TYPE ST_CycleData :
STRUCT
//-----------------------------------------------------------------------------------GENERAL------------------------------------------------------------------------------------//	

	nNest				: INT;
	bPass				: BOOL;
	bFail				: BOOL;	
	sDate				: STRING;	
	sTime				: STRING;
	
	LeakTest_Pass		: BOOL;
	LeakTest_Fail		: BOOL;
	
	Camera_Pass			: BOOL;
	Camera_Fail			: BOOL;
	
	//Height test
	
	LSS_ScaledHeight			: ARRAY [1..4] OF REAL;
	LSS_anSetPoint				: REAL;
	LSS_CalibrationHeight		: ARRAY [1..4] OF REAL;
	LSS_anRawMeasurement		: ARRAY [1..4] OF REAL;
	LSS_HeightPass				: ARRAY [1..4] OF BOOL;	
	LSS_HeightFail				: ARRAY [1..4] OF BOOL;	

	
	LSS_Pass			: BOOL;
	LSS_Fail			: BOOL;	

	
	//HMI, CSV
	sGeneralResult		: STRING;
	sCameraResult		: STRING;
	sHeightTestResult	: STRING;
	sLeakTesterResult	: STRING;
	
	sDistance1			: STRING;
	sDistance2			: STRING;
	sDistance3			: STRING;
	sDistance4			: STRING;
	
	sSetpoint1			: STRING;
	sSetpoint2			: STRING;
	sSetpoint3			: STRING;
	sSetpoint4			: STRING;
	
	

	
	


	
	
END_STRUCT
END_TYPE

(* stored: Version 1.1.0.1, ProductVersion 3.1.4026.18
   DUT ST_CycleData: Id {55f28d2e-fb51-4eb3-b909-a265f2991986} *)
